KUKA KRL data list: SetPlacePos.dat

&ACCESS RVO
&PARAM EDITMASK = *
DEFDAT SetPlacePos

ENDDAT
